Universal Robots PolyScope program: socket_hmi_example.urp

Program socket_hmi_example (installation=default directory=/ursim/programs createdIn=5.14.5 lastSavedIn=5.14.5 robotSerialNumber=20195599999)
Calibrated DH parameters: a=[0, -0.425, -0.3922, 0, 0, 0]; d=[0.1625, 0, 0, 0.1333, 0.0997, 0.0996]; alpha=[1.570796, 0, 0, 1.570796, -1.570796, 0]; deltaTheta=[0, 0, 0, 0, 0, 0]
InitVariablesNode
BeforeStart
  hmi_input := [0, 0, 0, 0]
  Timer (action=Start) variable(name=timer_1)
Robot Program (runOnlyOnce=false)
  If socket_open("192.168.87.42", 60000)
    Script: socket_send_string("Program running for " + to_str(timer_1) + " seconds")
    hmi_input := socket_read_binary_integer(3)
    Script: socket_close()
  Else 
    Popup Message (haltProgram=false message=Can't connect to HMI inputType=Text)
  'Run program sequence'
  Wait Sleep waitTime=5
